Fanuc KAREL source: NC0044.KL

-- PROVISIONAL review KL for V940-1; original PC SHA256 80c9319ca6fefe380a9be7814644655ae7e81d64a64e6e4c4def42bfdba54e8c
-- Incomplete behavior may be omitted. Consult companion uncertainty JSON. Do not deploy.
PROGRAM NC0044
%NOLOCKGROUP
-- UNRESOLVED_LOCAL_POOL 1 cells at code offset 3; source declarations unknown
-- DIRECT_LOCAL_WORD_ACCESS alone does not prove INTEGER, REAL, or BOOLEAN
BEGIN
  -- V9_CONDITION_STACK_HINT 2 bounded expression windows; static native code-base-relative target link; source arms held
  -- UNRESOLVED_PC offsets 0-8; opcodes 2B,2C,7B
  -- UNRESOLVED_PC offsets 13-20; opcodes 9D,23
  -- UNRESOLVED_PC offsets 25-38; opcodes 21,9D,57,79
  -- UNRESOLVED_PC offsets 43-60; opcodes 21,40,41,42
  -- UNRESOLVED_PC offsets 65-78; opcodes 21,9D,57,79
  -- UNRESOLVED_PC offsets 83-97; opcodes 21,9D,52,23
  -- UNRESOLVED_PC offsets 102-107; opcodes 7A
  -- UNRESOLVED_PC offsets 112-130; opcodes 21,2E,52,23
  -- UNRESOLVED_PC offsets 135-151; opcodes 7A,40,41,42
  -- UNRESOLVED_PC offsets 156-180; opcodes 21,2E,52,23,7A,43
  -- UNRESOLVED_PC offsets 185-203; opcodes 21,2E,52,23
  -- UNRESOLVED_PC offsets 213-218; opcodes 7A
  -- UNRESOLVED_PC offsets 223-241; opcodes 21,2E,52,23
  -- UNRESOLVED_PC offsets 251-255; opcodes 7F
  -- UNRESOLVED_PC offsets 260-264; opcodes 27,AA
  -- UNRESOLVED_PC offsets 269-273; opcodes 7F
END NC0044
